{attribute 'linkalways'} 
{attribute 'no_explicit_call' := 'This FB is a CLASS and must be accessed using methods or properties'}
{attribute 'enable_dynamic_creation'}
FUNCTION_BLOCK _FLOAT EXTENDS AliasDatatypeBase
VAR
	localData : FLOAT;
	activeData : REFERENCE TO FLOAT REF= localData;
	aliasBaseType : _LREAL(localData);
END_VAR

PROPERTY PUBLIC Address : PVOID
GET
Address := ADR(activeData);
END_GET
END_PROPERTY

METHOD PUBLIC ClearReference
VAR_INPUT
END_VAR
activeData REF= localData;
SetBaseTypeReference();
END_METHOD

METHOD PUBLIC Clone : I_Datatype
VAR
    pClone : POINTER TO _FLOAT;
END_VAR
pClone := __NEW(_FLOAT(InitialValue := Value));
Clone := pClone^;
END_METHOD

METHOD FB_init : BOOL
VAR_INPUT
	bInitRetains : BOOL; // if TRUE, the retain variables are initialized (warm start / cold start)
	bInCopyCode : BOOL;  // if TRUE, the instance afterwards gets moved into the copy code (online change)
	InitialValue : FLOAT;
END_VAR
localData := InitialValue;
SetBaseTypeReference();
AddBaseType(aliasBaseType);
END_METHOD

PROPERTY PUBLIC Identifier : T_MAXSTRING
GET
Identifier := 'FLOAT';
END_GET
END_PROPERTY

METHOD PUBLIC MakeReferenceTo
VAR_INPUT
	ReferenceTarget : REFERENCE TO FLOAT;
END_VAR
activeData REF= ReferenceTarget;
SetBaseTypeReference();
END_METHOD

METHOD PROTECTED SetBaseTypeReference
VAR_INPUT
END_VAR
aliasBaseType.MakeReferenceTo(activeData);
END_METHOD

PROPERTY PUBLIC Size : UDINT
GET
Size := SIZEOF(activeData);
END_GET
END_PROPERTY

METHOD TryMakeReferenceTo : BOOL
VAR_INPUT
	Target : I_Datatype;
END_VAR
VAR
	pTargetData : POINTER TO FLOAT;
END_VAR
IF NOT (Target.IecType = IecType) THEN
	RETURN;
END_IF

pTargetData := Target.Address;
activeData REF= pTargetData^;
SetBaseTypeReference();
TryMakeReferenceTo := TRUE;
END_METHOD

PROPERTY PUBLIC Value : FLOAT
GET
Value := activeData;
END_GET
SET
activeData := Value;
END_SET
END_PROPERTY

END_FUNCTION_BLOCK

(* stored: Version 1.1.0.1, ProductVersion 3.1.4024.12
   POU _FLOAT: Id {e544e036-9c3a-0a61-3910-dde23db4424d}, SpecialFunc None
   Folder Constructor: Id {8c9565a5-0beb-0708-11b9-437c7905f40f}
   Folder Protected: Id {89712a52-18ae-07b8-3966-fea83bf3efd8}
   Property Address: Id {78bf8f79-e163-0fd5-39ad-6ee17491b8ab}
   Get Get: Id {b4d73089-202a-0273-0cf1-5ca22886a16e}
   Method ClearReference: Id {7ff94cd1-223a-0f69-0142-804d3b7d702e}
   Method Clone: Id {80e0ab70-36a0-0025-1259-7c61c0c1d70a}
   Method FB_init: Id {be4b5ada-bdcb-07bb-1be4-38c060ad099b}
   Property Identifier: Id {f104ef4a-6158-01ae-0dab-342a586715c3}
   Get Get: Id {45ee9c3d-5b78-0d3b-0f19-9712248ecc92}
   Method MakeReferenceTo: Id {07b05c37-a2e3-05b9-0eef-db713695e8b2}
   Method SetBaseTypeReference: Id {841b5ad7-ce87-08eb-1d96-dac4d62db896}
   Property Size: Id {f340fa22-61d4-09f1-3c07-c59f10ec7f1f}
   Get Get: Id {c57484b6-63dc-06b7-2e00-11f44e37a19b}
   Method TryMakeReferenceTo: Id {c1df8b2c-bcae-024b-3fa1-2aa3bb02b580}
   Property Value: Id {657e324f-08a8-01cd-3aae-f90fbe8b24be}
   Get Get: Id {749b3910-41db-0ef2-0bfa-518471ca9a45}
   Set Set: Id {7c81c33a-57a7-0b4d-05db-d1391735f373} *)
